// TIA Portal V18 export
FUNCTION_BLOCK "SR_TRIG"   // FB34, FBD
{ S7_Optimized_Access := 'TRUE' }
VERSION : 0.1
// stored: AutoNumber true, IsIECCheckEnabled false, IsRetainMemResEnabled false, MemoryReserve 100, SetENOAutomatically false, UDAEnableTagReadback false
   VAR_INPUT
      SR_CNTRL : Bool;
   END_VAR
   VAR_IN_OUT
      Q : Bool;
   END_VAR
   VAR
      mem1 : Bool;
      mem2 : Bool;
   END_VAR
   VAR_TEMP   // added for the SCL form of the ladder/FBD networks
      _w1 : Bool;
      _w2 : Bool;
   END_VAR
BEGIN

REGION Network 1
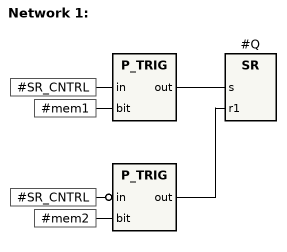
   #_w1 := #SR_CNTRL AND NOT #mem1;   // rising edge
   #mem1 := #SR_CNTRL;
   #_w2 := NOT #SR_CNTRL AND NOT #mem2;   // rising edge
   #mem2 := NOT #SR_CNTRL;
   IF #_w1 THEN
       #Q := TRUE;   // SR flip-flop
   END_IF;
   IF #_w2 THEN #Q := FALSE; END_IF;
END_REGION
END_FUNCTION_BLOCK
